FUNCTION_BLOCK AUI_TO_ALR (* Composite FB for converting AUI (UINT) adapter to ALR (LREAL) adapter *)
  (* Standard: 61499-2; Description: Copyright (c) 2026 HR Agrartechnik GmbH This program and the accompanying materials are made available under the terms of the Eclipse Public License 2.0 which is available at https://www.eclipse.org/legal/epl-2.0/ SPDX-License-Identifier: EPL-2.0 *)
  (* Version 1.0, 2026-02-17, Franz Höpfinger, HR Agrartechnik GmbH *)
  PACKAGE adapter::conversion::unidirectional;
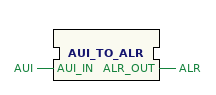
  SOCKETS
    AUI_IN : adapter::types::unidirectional::AUI; (* UINT Adapter Input *)
  END_SOCKETS
  PLUGS
    ALR_OUT : adapter::types::unidirectional::ALR; (* LREAL Adapter Output *)
  END_PLUGS
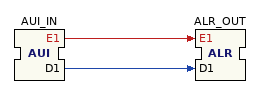
  EVENT_CONNECTIONS
    AUI_IN.E1 TO ALR_OUT.E1;
  END_CONNECTIONS
  DATA_CONNECTIONS
    AUI_IN.D1 TO ALR_OUT.D1;
  END_CONNECTIONS
END_FUNCTION_BLOCK
